Fanuc KAREL source: kb00018.KL

-- PROVISIONAL review KL for V1013-1; original PC SHA256 c511c0f821a85117aed6a27652ae159bc10d67d422a0c745412cd1fc557d5ef0
-- Incomplete behavior may be omitted. Consult companion uncertainty JSON. Do not deploy.
PROGRAM KB00018
%NOLOCKGROUP
BEGIN
  -- UNRESOLVED_PC offsets 5-12; opcodes 9D,23
  -- UNRESOLVED_PC offsets 17-65; opcodes 27,22,1C,22,1C,22,1C,22,27,9D,31
  -- UNRESOLVED_PC offsets 70-74; opcodes 7F
END KB00018
